Yaskawa INFORM job: TEST_HOLES.JBI

/JOB
//NAME TEST_HOLES
///FOLDERNAME INNE
//POS
///NPOS 4,4,4,0,0,0
///TOOL 0
///POSTYPE PULSE
///PULSE
C00000=-113507,-92089,-39731,-55954,55727,-71701
C00001=-115316,-71951,-32153,-52991,58136,-74596
C00002=-123662,-34022,-14256,-44914,58876,-80336
C00003=-134148,-129577,-50186,-64382,36705,-69645
BC00000=363517,7680,447965
BC00001=363517,7680,447965
BC00002=363517,7680,447965
BC00003=363517,7680,447965
EC00000=0,0
EC00001=0,0
EC00002=0,0
EC00003=0,0
//INST
///DATE 2023/10/04 15:16
///ATTR SC,RW
///GROUP1 RB1,BS1
///GROUP2 ST1
NOP
'test_holes
MOVJ C00000 BC00000 VJ=100.00  +MOVJ EC00000 VJ=100.00
MOVJ C00001 BC00001 VJ=100.00  +MOVJ EC00001 VJ=100.00
MOVJ C00002 BC00002 VJ=100.00  +MOVJ EC00002 VJ=100.00
MOVJ C00003 BC00003 VJ=100.00  +MOVJ EC00003 VJ=100.00
END
